(* IEC 61131-3 sources: ConveyorControl-with-PLC/4E_Gruppe1_Graf_Projekt1/Class/class0, 1 file *)

(* ---- class0.st ---- *)
(*!
<Class
	Name               = "class0"
	Revision           = "0.0"
	RealtimeTask       = "false"
	CyclicTask         = "false"
	DefCyclictime      = "10 ms"
	BackgroundTask     = "false"
	Sigmatek           = "false"
	OSInterface        = "false"
	HighPriority       = "false"
	Automatic          = "false"
	UpdateMode         = "Prescan"
	SharedCommandTable = "true"
	Objectsize         = "(284,120)">
	<Channels>
		<Server Name="ClassSvr" Visualized="false" Initialize="false" WriteProtected="true" Retentive="false"/>
		<Server Name="counter" Visualized="false" Initialize="false" WriteProtected="false" Retentive="false"/>
		<Server Name="hmiLight" Visualized="true" Initialize="false" WriteProtected="false" Retentive="false"/>
		<Server Name="hmiStart" Visualized="true" Initialize="false" WriteProtected="false" Retentive="false"/>
		<Server Name="ssw" Visualized="false" Initialize="false" WriteProtected="false" Retentive="false"/>
		<Client Name="CYL" Required="true" Internal="false"/>
		<Client Name="lightbarrier" Required="true" Internal="false"/>
		<Client Name="MTR" Required="true" Internal="false"/>
		<Client Name="StartBTN" Required="true" Internal="false"/>
	</Channels>
</Class>
*)
class0 : CLASS
	TYPE
	  _steps :  //! <Type Public="true" Name="_steps"/>
	  (
	    wait4start,
	    wait4light,
	    wait4time
	  )$UDINT;
	END_TYPE
  //Servers:
	ClassSvr 	: SvrChCmd_DINT;
	ssw 	: SvrCh__steps_PTofCls_class0;
	counter 	: SvrCh_DINT;
	hmiStart 	: SvrCh_DINT;
	hmiLight 	: SvrCh_DINT;
  //Clients:
	MTR 	: CltCh_DINT;
	StartBTN 	: CltCh_DINT;
	lightbarrier 	: CltCh_DINT;
	CYL 	: CltCh_DINT;
  //Variables:
  //Functions:

	FUNCTION VIRTUAL GLOBAL CyWork
		VAR_INPUT
			EAX 	: UDINT;
		END_VAR
		VAR_OUTPUT
			state (EAX) 	: UDINT;
		END_VAR;
  //Tables:
	FUNCTION @STD
		VAR_OUTPUT
			ret_code	: CONFSTATES;
		END_VAR;
	FUNCTION GLOBAL TAB @CT_;
END_CLASS;

FUNCTION VIRTUAL GLOBAL class0::CyWork
	VAR_INPUT
		EAX 	: UDINT;
	END_VAR
	VAR_OUTPUT
		state (EAX) 	: UDINT;
	END_VAR

  StartBTN := StartBTN.Read();
  lightbarrier := lightbarrier.Read();

  case ssw of

  wait4start:

    if StartBTN = 1 then
      MTR := 1;
      ssw := wait4light;
    end_if;

  wait4light:

    if lightbarrier = 1 then
      MTR := 0;
      CYL := 1;
      ssw := wait4time;
    end_if;

  wait4time:

     if counter = 700 then
      CYL := 0;
      counter := 0;
      ssw := wait4start;
     else
      counter += 1;
     end_if;

  end_case;

  MTR.Write (MTR);
  CYL.Write (CYL);

	state := READY;

END_FUNCTION
